Universal Robots PolyScope program: y_force.urp

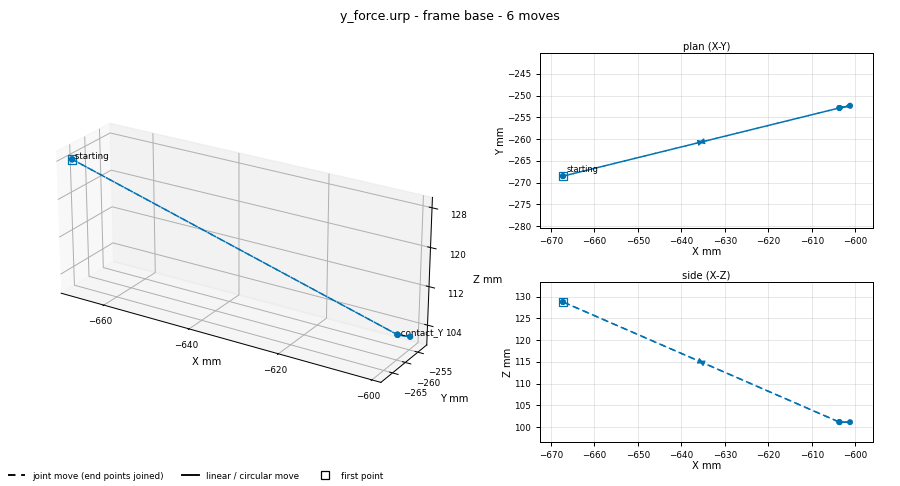
[picture p0: tool path of y_force.urp in frame base, 6 of 6 moves have a stored position in this frame; points joined in program order, loops and branches not executed]
Program y_force_mh (installation=weiss_default directory=/programs/usbdisk_0/Max_MA createdIn=5.12.4 lastSavedIn=5.14.3 robotSerialNumber=20235500024)
Calibrated DH parameters: a=[0.000122, -0.425124, -0.373197, -0.000038, 0.000163, 0]; d=[0.162581, -17.281615, 1.061906, 16.353116, 0.099729, 0.099553]; alpha=[1.570231, 0.000934, 0.007511, 1.569966, -1.569202, 0]; deltaTheta=[0, -0.037947, -0.277584, 0.315538, 0.000001, -0.000001]
InitVariablesNode
BeforeStart
  Script: socket_close("DataSocket")
  Script: connected = socket_open("192.168.100.0",30000,"DataSocket")
  force_measure := False
  If connected ≟  False (checkContinuously=true)
    Halt
Robot Program (runOnlyOnce=true)
  MoveJ speed 60 deg/s, acceleration 80 deg/s^2 (useActiveTCP=true) feature=Base
    Waypoint starting: TCP in base x=-667.239 y=-268.524 z=128.773 mm, rx=0.3939 ry=-3.1168 rz=-0.0001 rad; joints [11.313, -53.135, 79.364, -116.139, -89.581, -93.029] deg; TCP offset x=0 y=0 z=100 mm, rx=0 ry=0 rz=0 rad
    SuppressedNode
      Set DigitalOutput pin=digital_out[0]; digitalValue=1
    Timer (action=Start) variable(name=timer_1)
    Timer (action=Start) variable(name=timer_3)
    Waypoint contact_Y: TCP in base x=-603.671 y=-252.842 z=101.144 mm, rx=0.3485 ry=-3.1219 rz=-0.0001 rad; joints [11.043, -58.892, 93.878, -124.915, -89.601, -91.571] deg
    SuppressedNode
      Waypoint contact_l_width: TCP in base x=-639.916 y=-260.393 z=101.315 mm, rx=0.3486 ry=-3.1219 rz=0 rad; joints [11.085, -54.741, 86.742, -121.927, -89.588, -91.553] deg
    SuppressedNode
      Waypoint contact_xl_widt: TCP in base x=-640.842 y=-260.602 z=101.034 mm, rx=0.3486 ry=-3.1218 rz=-0.0001 rad; joints [11.088, -54.614, 86.571, -121.891, -89.59, -91.55] deg
    SuppressedNode
      Waypoint contact_s_width: TCP in base x=-636.868 y=-259.715 z=101.666 mm, rx=0.3487 ry=-3.1218 rz=-0.0001 rad; joints [11.078, -55.125, 87.348, -122.152, -89.59, -91.56] deg
    SuppressedNode
      Waypoint contact_xs_widt: TCP in base x=-635.864 y=-259.478 z=101.654 mm, rx=0.3487 ry=-3.1219 rz=0 rad; joints [11.074, -55.242, 87.552, -122.237, -89.59, -91.563] deg
    SuppressedNode
      Waypoint contact_y_36mm: TCP in base x=-636.451 y=-259.648 z=95.642 mm, rx=0.3487 ry=-3.1218 rz=-0.0001 rad; joints [11.078, -54.733, 87.711, -122.906, -89.591, -91.555] deg
    force_measure := True
    Loop Counting (count=10) loopVariable(name=Loop_3)
      MoveL speed 3 mm/s, acceleration 600 mm/s^2 (useActiveTCP=true) feature=Base
        Waypoint displ_25mmm: TCP in base x=-601.234 y=-252.341 z=101.139 mm, rx=0.3486 ry=-3.1218 rz=-0.0001 rad; joints [11.04, -59.167, 94.342, -125.105, -89.6, -91.578] deg
        SuppressedNode
          Waypoint displ_s_width: TCP in base x=-632.989 y=-258.827 z=101.671 mm, rx=0.3486 ry=-3.1218 rz=0 rad; joints [11.067, -55.58, 88.136, -122.486, -89.59, -91.568] deg
        SuppressedNode
          Waypoint displ_l_width: TCP in base x=-637.978 y=-259.975 z=101.363 mm, rx=0.3488 ry=-3.1218 rz=-0.0002 rad; joints [11.083, -54.973, 87.137, -122.097, -89.596, -91.559] deg
        SuppressedNode
          Waypoint displ_2_xl_w: TCP in base x=-639.326 y=-260.245 z=100.991 mm, rx=0.3486 ry=-3.1218 rz=0 rad; joints [11.082, -54.789, 86.882, -122.025, -89.589, -91.553] deg
        SuppressedNode
          Waypoint displ_xs_width: TCP in base x=-632.947 y=-258.844 z=101.701 mm, rx=0.3488 ry=-3.1218 rz=0 rad; joints [11.069, -55.587, 88.142, -122.488, -89.59, -91.57] deg
        SuppressedNode
          Waypoint displ5mml30: TCP in base x=-631.496 y=-258.529 z=89.644 mm, rx=0.3487 ry=-3.1219 rz=-0.0001 rad; joints [11.064, -54.858, 88.979, -124.049, -89.593, -91.561] deg
        SuppressedNode
          Waypoint displ5mm36: TCP in base x=-631.558 y=-258.54 z=95.654 mm, rx=0.3487 ry=-3.1218 rz=-0.0001 rad; joints [11.066, -55.302, 88.701, -123.328, -89.594, -91.564] deg
        SuppressedNode
          Waypoint displ5mm48: TCP in base x=-632.874 y=-258.835 z=107.651 mm, rx=0.3486 ry=-3.1219 rz=0 rad; joints [11.07, -56.023, 87.864, -121.77, -89.588, -91.57] deg
        SuppressedNode
          Waypoint displ5mm54: TCP in base x=-633.423 y=-258.929 z=113.711 mm, rx=0.3486 ry=-3.1217 rz=-0.0001 rad; joints [11.071, -56.388, 87.453, -121, -89.591, -91.574] deg
        SuppressedNode
          Waypoint contact_xs_widt: TCP in base x=-635.864 y=-259.478 z=101.654 mm, rx=0.3487 ry=-3.1219 rz=0 rad; joints [11.074, -55.242, 87.552, -122.237, -89.59, -91.563] deg
        Waypoint contact_Y: TCP in base x=-603.671 y=-252.842 z=101.144 mm, rx=0.3485 ry=-3.1219 rz=-0.0001 rad; joints [11.043, -58.892, 93.878, -124.915, -89.601, -91.571] deg
        SuppressedNode
          Waypoint contact_l_width: TCP in base x=-639.916 y=-260.393 z=101.315 mm, rx=0.3486 ry=-3.1219 rz=0 rad; joints [11.085, -54.741, 86.742, -121.927, -89.588, -91.553] deg
        SuppressedNode
          Waypoint contact_xl_widt: TCP in base x=-640.842 y=-260.602 z=101.034 mm, rx=0.3486 ry=-3.1218 rz=-0.0001 rad; joints [11.088, -54.614, 86.571, -121.891, -89.59, -91.55] deg
        SuppressedNode
          Waypoint contact_s_width: TCP in base x=-636.868 y=-259.715 z=101.666 mm, rx=0.3487 ry=-3.1218 rz=-0.0001 rad; joints [11.078, -55.125, 87.348, -122.152, -89.59, -91.56] deg
        SuppressedNode
          Waypoint contact_y_36mm: TCP in base x=-636.451 y=-259.648 z=95.642 mm, rx=0.3487 ry=-3.1218 rz=-0.0001 rad; joints [11.078, -54.733, 87.711, -122.906, -89.591, -91.555] deg
        SuppressedNode
          Waypoint contact_y_36mm: TCP in base x=-636.451 y=-259.648 z=95.642 mm, rx=0.3487 ry=-3.1218 rz=-0.0001 rad; joints [11.078, -54.733, 87.711, -122.906, -89.591, -91.555] deg
        SuppressedNode
          Waypoint contact_y_48: TCP in base x=-637.767 y=-259.922 z=107.69 mm, rx=0.3486 ry=-3.1218 rz=-0.0001 rad; joints [11.082, -55.449, 86.874, -121.357, -89.589, -91.561] deg
        SuppressedNode
          Waypoint contact_y_54: TCP in base x=-638.275 y=-260.032 z=113.701 mm, rx=0.3486 ry=-3.1218 rz=-0.0001 rad; joints [11.085, -55.808, 86.464, -120.587, -89.591, -91.564] deg
        SuppressedNode
          Waypoint Waypoint_1: TCP in base x=-582.371 y=-248.401 z=111.231 mm, rx=0.3487 ry=-3.122 rz=0 rad; joints [11.016, -62.09, 97.362, -125.193, -89.601, -91.604] deg
    force_measure := False
    Waypoint contact_Y: TCP in base x=-603.671 y=-252.842 z=101.144 mm, rx=0.3485 ry=-3.1219 rz=-0.0001 rad; joints [11.043, -58.892, 93.878, -124.915, -89.601, -91.571] deg
    SuppressedNode
      Waypoint contact_xs_widt: TCP in base x=-635.864 y=-259.478 z=101.654 mm, rx=0.3487 ry=-3.1219 rz=0 rad; joints [11.074, -55.242, 87.552, -122.237, -89.59, -91.563] deg
    SuppressedNode
      Waypoint contact_s_width: TCP in base x=-636.868 y=-259.715 z=101.666 mm, rx=0.3487 ry=-3.1218 rz=-0.0001 rad; joints [11.078, -55.125, 87.348, -122.152, -89.59, -91.56] deg
    SuppressedNode
      Waypoint contact_l_width: TCP in base x=-639.916 y=-260.393 z=101.315 mm, rx=0.3486 ry=-3.1219 rz=0 rad; joints [11.085, -54.741, 86.742, -121.927, -89.588, -91.553] deg
    SuppressedNode
      Waypoint contact_xl_widt: TCP in base x=-640.842 y=-260.602 z=101.034 mm, rx=0.3486 ry=-3.1218 rz=-0.0001 rad; joints [11.088, -54.614, 86.571, -121.891, -89.59, -91.55] deg
    SuppressedNode
      Waypoint contact_y_36mm: TCP in base x=-636.451 y=-259.648 z=95.642 mm, rx=0.3487 ry=-3.1218 rz=-0.0001 rad; joints [11.078, -54.733, 87.711, -122.906, -89.591, -91.555] deg
    Wait Sleep waitTime=2
    Timer (action=Stop) variable=timer_3
    Timer (action=Reset) variable=timer_3
    SuppressedNode
      Wait Sleep waitTime=5
    Timer (action=Stop) variable=timer_1
    Waypoint starting: TCP in base x=-667.239 y=-268.524 z=128.773 mm, rx=0.3939 ry=-3.1168 rz=-0.0001 rad; joints [11.313, -53.135, 79.364, -116.139, -89.581, -93.029] deg
Thread Thread_1 (runOnlyOnce=false)
  If force_measure ≟ True
    counter := 1
    SuppressedNode
      Wait Sleep waitTime=1
    Timer (action=Reset) variable(name=timer_2)
    Timer (action=Start) variable=timer_2
    Loop While (checkContinuously=true) expression=force_measure ≟  True
      force_value := get_tcp_force()
      pos_value := get_actual_tcp_pose()
      SuppressedNode
        msg_out := [timer_2,force_value[0],force_value[1],force_value[2],force_value[3],force_value[4],force_value[5]]
      msg_out := [timer_2,force_value[0],force_value[1],force_value[2],force_value[3],force_value[4],force_value[5],pos_value[0],pos_value[1],pos_value[2],pos_value[3],pos_value[4],pos_value[5]]
      Script: socket_send_string(msg_out,"DataSocket")
      SuppressedNode
        Script: data = socket_read_ascii_float(1,"DataSocket")
      SuppressedNode
        screw_force_lim := data[1]
      counter := counter + 1
      Wait Sleep waitTime=0.02
    Script: socket_send_string("end","DataSocket")
    Wait Sleep waitTime=0.01
    Script: socket_close("DataSocket")
    Timer (action=Stop) variable=timer_2
SuppressedNode
  Thread Thread_2 (runOnlyOnce=false)
    URCap Gripper Activate (Robotiq_Grippers, Robotiq Inc.) dataModel(ResetAndActivateKey=true)
    URCap GRIPKIT Reference (GRIPKIT by Weiss Robotics, Weiss Robotics GmbH & Co. KG) dataModel(reference1=true)
